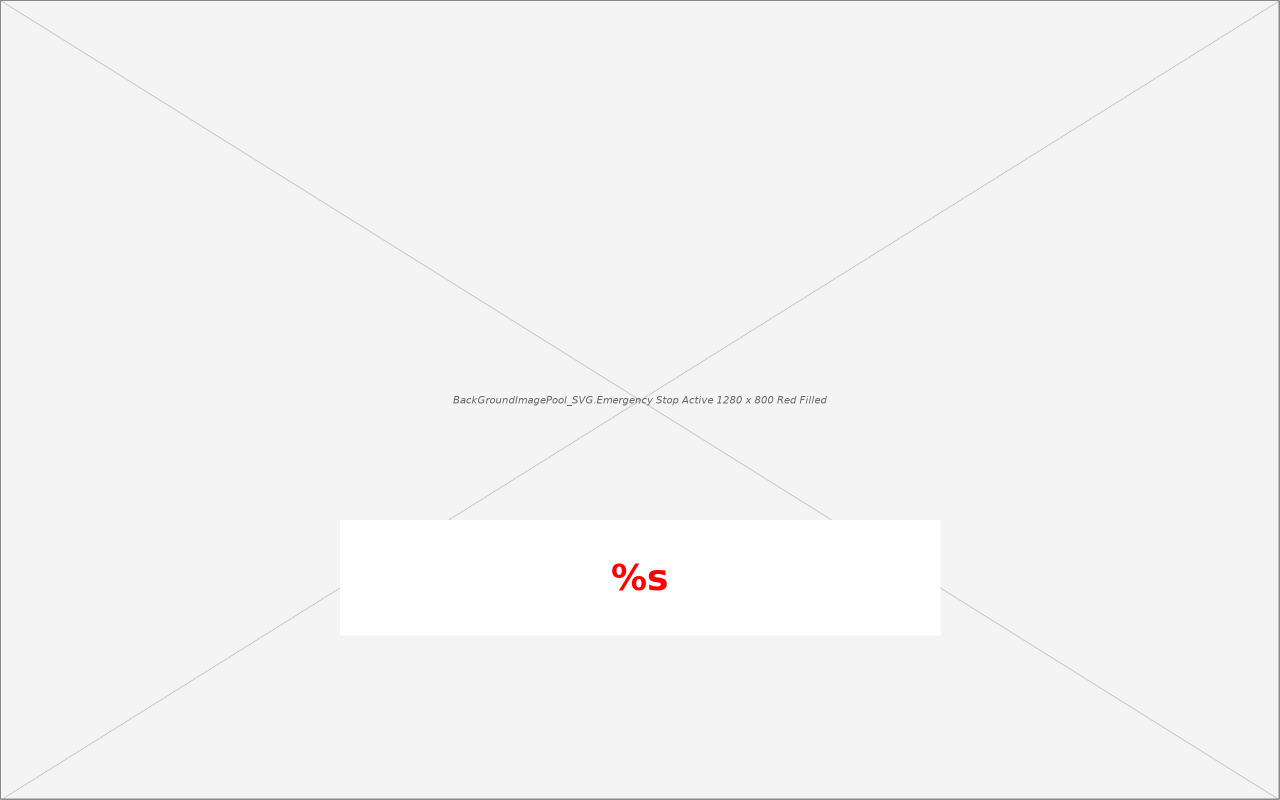
VISUALIZATION BG_Emergency  // 1280x800
VAR_IN_OUT
	sMessage : STRING;
END_VAR
    Image (0,0 1280x800), invisible if: NOT GVL_HMI.fbHMIControl.bShowEmergencyOverlay, image: BackGroundImagePool_SVG.Emergency Stop Active 1280 x 800 Red Filled
    Textfield (340,520 600x115), "%s", text variable: sMessage
END_VISUALIZATION

(* stored: Version 1.1.0.1, ProductVersion 3.1.4024.11
   Visu BG_Emergency: Id {2f5e5ddc-e4de-47b5-8b36-ec044437ab0c} *)
